// TIA Portal V17 export
// export: Created 2023-08-28T22:41:32.6164324Z, ExportSetting WithDefaults, DisplayName Totally Integrated Automation Portal, DisplayVersion V17 Update 5, DisplayName TIA Portal Openness, DisplayVersion V17 Update 5, DisplayName TIA Portal Teamcenter Gateway, DisplayVersion V17 Update 5, DisplayName TIA Portal Version Control Interface, DisplayVersion V17, DisplayName Simotion SCOUT TIA, DisplayVersion 5.4.3.0, DisplayName TIA Portal Test Suite Advanced, DisplayVersion V17 Update 1, DisplayName SIMOCODE ES, DisplayVersion V17 Update 5, DisplayName SINAMICS Startdrive Advanced, DisplayVersion V17 SP1, DisplayName SINAMICS Startdrive G130, G150, S120, S150, SINAMICS MV, S210, DisplayVersion V17 SP1, DisplayName SINAMICS Startdrive G110M, G120, G120C, G120D, G120P, G115D, DisplayVersion V17 SP1, DisplayName SIRIUS Safety ES, DisplayVersion V17 Update 5, DisplayName STEP 7 Professional, DisplayVersion V17 Update 5, DisplayName STEP 7 CFC, DisplayVersion V17 Update 1, DisplayName STEP 7 Safety, DisplayVersion V17, DisplayName WinCC Advanced, DisplayVersion V17 Update 5, DisplayName SIMATIC Visualization Architect, DisplayVersion V17 Update 5
DATA_BLOCK "FDBK_Error_n0015-uc16-el001-k30001_SN50_1"   // DB2000, F_DB
// stored: AutoNumber true, DBAccessibleFromOPCUA true, DBAccessibleFromWebserver true, InstanceOfName 03_FDBACK error, InstanceOfType FB
"03_FDBACK error "
BEGIN
END_DATA_BLOCK

DATA_BLOCK "FDBK_Error_n0015-uc16-el001-k30001_SN50_2"   // DB2001, F_DB
// stored: AutoNumber true, DBAccessibleFromOPCUA true, DBAccessibleFromWebserver true, InstanceOfName 03_FDBACK error, InstanceOfType FB
"03_FDBACK error "
BEGIN
END_DATA_BLOCK

DATA_BLOCK "FDBK_Error_n0015-uc16-el001-k30001_SN50_3"   // DB2002, F_DB
// stored: AutoNumber true, DBAccessibleFromOPCUA true, DBAccessibleFromWebserver true, InstanceOfName 03_FDBACK error, InstanceOfType FB
"03_FDBACK error "
BEGIN
END_DATA_BLOCK

DATA_BLOCK "FDBK_Error_n0017-lv004-el001-k30001_SN50_1"   // DB2003, F_DB
// stored: AutoNumber true, DBAccessibleFromOPCUA true, DBAccessibleFromWebserver true, InstanceOfName 03_FDBACK error, InstanceOfType FB
"03_FDBACK error "
BEGIN
END_DATA_BLOCK

DATA_BLOCK "FDBK_Error_n0018-lv004-el001-k30001_SN50_1"   // DB2004, F_DB
// stored: AutoNumber true, DBAccessibleFromOPCUA true, DBAccessibleFromWebserver true, InstanceOfName 03_FDBACK error, InstanceOfType FB
"03_FDBACK error "
BEGIN
END_DATA_BLOCK

DATA_BLOCK "FDBK_Error_n0020-uc15-el001-k30001_SN50_1"   // DB2005, F_DB
// stored: AutoNumber true, DBAccessibleFromOPCUA true, DBAccessibleFromWebserver true, InstanceOfName 03_FDBACK error, InstanceOfType FB
"03_FDBACK error "
BEGIN
END_DATA_BLOCK

DATA_BLOCK "FDBK_Error_n0020-uc15-el001-k30001_SN50_2"   // DB2006, F_DB
// stored: AutoNumber true, DBAccessibleFromOPCUA true, DBAccessibleFromWebserver true, InstanceOfName 03_FDBACK error, InstanceOfType FB
"03_FDBACK error "
BEGIN
END_DATA_BLOCK

DATA_BLOCK "FDBK_Error_n0020-uc15-el001-k30001_SN50_3"   // DB2007, F_DB
// stored: AutoNumber true, DBAccessibleFromOPCUA true, DBAccessibleFromWebserver true, InstanceOfName 03_FDBACK error, InstanceOfType FB
"03_FDBACK error "
BEGIN
END_DATA_BLOCK

DATA_BLOCK "FDBK_Error_n0021-icg11-el001-k30001_SN50_1"   // DB2008, F_DB
// stored: AutoNumber true, DBAccessibleFromOPCUA true, DBAccessibleFromWebserver true, InstanceOfName 03_FDBACK error, InstanceOfType FB
"03_FDBACK error "
BEGIN
END_DATA_BLOCK

DATA_BLOCK "FDBK_Error_n0022-icg21-el001-k30001_SN50_1"   // DB2009, F_DB
// stored: AutoNumber true, DBAccessibleFromOPCUA true, DBAccessibleFromWebserver true, InstanceOfName 03_FDBACK error, InstanceOfType FB
"03_FDBACK error "
BEGIN
END_DATA_BLOCK

DATA_BLOCK "FDBK_Error_n0025-uc14-el001-k30001_SN50_1"   // DB2010, F_DB
// stored: AutoNumber true, DBAccessibleFromOPCUA true, DBAccessibleFromWebserver true, InstanceOfName 03_FDBACK error, InstanceOfType FB
"03_FDBACK error "
BEGIN
END_DATA_BLOCK

DATA_BLOCK "FDBK_Error_n0025-uc14-el001-k30001_SN50_2"   // DB2011, F_DB
// stored: AutoNumber true, DBAccessibleFromOPCUA true, DBAccessibleFromWebserver true, InstanceOfName 03_FDBACK error, InstanceOfType FB
"03_FDBACK error "
BEGIN
END_DATA_BLOCK

DATA_BLOCK "FDBK_Error_n0025-uc14-el001-k30001_SN50_3"   // DB2012, F_DB
// stored: AutoNumber true, DBAccessibleFromOPCUA true, DBAccessibleFromWebserver true, InstanceOfName 03_FDBACK error, InstanceOfType FB
"03_FDBACK error "
BEGIN
END_DATA_BLOCK

DATA_BLOCK "FDBK_Error_n0039-lv001-el001-k30001_SN50_1"   // DB2013, F_DB
// stored: AutoNumber true, DBAccessibleFromOPCUA true, DBAccessibleFromWebserver true, InstanceOfName 03_FDBACK error, InstanceOfType FB
"03_FDBACK error "
BEGIN
END_DATA_BLOCK

DATA_BLOCK "FDBK_Error_n0040-lv001-el001-k30001_SN50_1"   // DB2014, F_DB
// stored: AutoNumber true, DBAccessibleFromOPCUA true, DBAccessibleFromWebserver true, InstanceOfName 03_FDBACK error, InstanceOfType FB
"03_FDBACK error "
BEGIN
END_DATA_BLOCK

DATA_BLOCK "FDBK_Error_n0041-uf31-el002-k30001_SN50_1"   // DB2015, F_DB
// stored: AutoNumber true, DBAccessibleFromOPCUA true, DBAccessibleFromWebserver true, InstanceOfName 03_FDBACK error, InstanceOfType FB
"03_FDBACK error "
BEGIN
END_DATA_BLOCK

DATA_BLOCK "FDBK_Error_n0042-uf41-el002-k30001_SN50_1"   // DB2016, F_DB
// stored: AutoNumber true, DBAccessibleFromOPCUA true, DBAccessibleFromWebserver true, InstanceOfName 03_FDBACK error, InstanceOfType FB
"03_FDBACK error "
BEGIN
END_DATA_BLOCK

DATA_BLOCK "FDBK_Error_n0044-ct1-el001-k30001_SN50_1"   // DB2017, F_DB
// stored: AutoNumber true, DBAccessibleFromOPCUA true, DBAccessibleFromWebserver true, InstanceOfName 03_FDBACK error, InstanceOfType FB
"03_FDBACK error "
BEGIN
END_DATA_BLOCK

DATA_BLOCK "FDBK_Error_n0045-ct1-el002-k30001_SN50_1"   // DB2018, F_DB
// stored: AutoNumber true, DBAccessibleFromOPCUA true, DBAccessibleFromWebserver true, InstanceOfName 03_FDBACK error, InstanceOfType FB
"03_FDBACK error "
BEGIN
END_DATA_BLOCK

DATA_BLOCK "FDBK_Error_n0046-ct1-el003-k30001_SN50_1"   // DB2019, F_DB
// stored: AutoNumber true, DBAccessibleFromOPCUA true, DBAccessibleFromWebserver true, InstanceOfName 03_FDBACK error, InstanceOfType FB
"03_FDBACK error "
BEGIN
END_DATA_BLOCK

DATA_BLOCK "FDBK_Error_n0047-lv002-el001-k30001_SN50_1"   // DB2020, F_DB
// stored: AutoNumber true, DBAccessibleFromOPCUA true, DBAccessibleFromWebserver true, InstanceOfName 03_FDBACK error, InstanceOfType FB
"03_FDBACK error "
BEGIN
END_DATA_BLOCK

DATA_BLOCK "FDBK_Error_n0048-lv002-el001-k30001_SN50_1"   // DB2021, F_DB
// stored: AutoNumber true, DBAccessibleFromOPCUA true, DBAccessibleFromWebserver true, InstanceOfName 03_FDBACK error, InstanceOfType FB
"03_FDBACK error "
BEGIN
END_DATA_BLOCK

DATA_BLOCK "FDBK_Error_n0050-uc13-el001-k30001_SN50_1"   // DB2022, F_DB
// stored: AutoNumber true, DBAccessibleFromOPCUA true, DBAccessibleFromWebserver true, InstanceOfName 03_FDBACK error, InstanceOfType FB
"03_FDBACK error "
BEGIN
END_DATA_BLOCK

DATA_BLOCK "FDBK_Error_n0050-uc13-el001-k30001_SN50_2"   // DB2023, F_DB
// stored: AutoNumber true, DBAccessibleFromOPCUA true, DBAccessibleFromWebserver true, InstanceOfName 03_FDBACK error, InstanceOfType FB
"03_FDBACK error "
BEGIN
END_DATA_BLOCK

DATA_BLOCK "FDBK_Error_n0050-uc13-el001-k30001_SN50_3"   // DB2024, F_DB
// stored: AutoNumber true, DBAccessibleFromOPCUA true, DBAccessibleFromWebserver true, InstanceOfName 03_FDBACK error, InstanceOfType FB
"03_FDBACK error "
BEGIN
END_DATA_BLOCK

DATA_BLOCK "FDBK_Error_n0053-uc12-el001-k30001_SN50_1"   // DB2025, F_DB
// stored: AutoNumber true, DBAccessibleFromOPCUA true, DBAccessibleFromWebserver true, InstanceOfName 03_FDBACK error, InstanceOfType FB
"03_FDBACK error "
BEGIN
END_DATA_BLOCK

DATA_BLOCK "FDBK_Error_n0053-uc12-el001-k30001_SN50_2"   // DB2026, F_DB
// stored: AutoNumber true, DBAccessibleFromOPCUA true, DBAccessibleFromWebserver true, InstanceOfName 03_FDBACK error, InstanceOfType FB
"03_FDBACK error "
BEGIN
END_DATA_BLOCK

DATA_BLOCK "FDBK_Error_n0053-uc12-el001-k30001_SN50_3"   // DB2027, F_DB
// stored: AutoNumber true, DBAccessibleFromOPCUA true, DBAccessibleFromWebserver true, InstanceOfName 03_FDBACK error, InstanceOfType FB
"03_FDBACK error "
BEGIN
END_DATA_BLOCK

DATA_BLOCK "FDBK_Error_n0054-uf31-el003-k30001_SN50_1"   // DB2028, F_DB
// stored: AutoNumber true, DBAccessibleFromOPCUA true, DBAccessibleFromWebserver true, InstanceOfName 03_FDBACK error, InstanceOfType FB
"03_FDBACK error "
BEGIN
END_DATA_BLOCK

DATA_BLOCK "FDBK_Error_n0057-uc11-el001-k30001_SN50_1"   // DB2029, F_DB
// stored: AutoNumber true, DBAccessibleFromOPCUA true, DBAccessibleFromWebserver true, InstanceOfName 03_FDBACK error, InstanceOfType FB
"03_FDBACK error "
BEGIN
END_DATA_BLOCK

DATA_BLOCK "FDBK_Error_n0057-uc11-el001-k30001_SN50_2"   // DB2030, F_DB
// stored: AutoNumber true, DBAccessibleFromOPCUA true, DBAccessibleFromWebserver true, InstanceOfName 03_FDBACK error, InstanceOfType FB
"03_FDBACK error "
BEGIN
END_DATA_BLOCK

DATA_BLOCK "FDBK_Error_n0057-uc11-el001-k30001_SN50_3"   // DB2031, F_DB
// stored: AutoNumber true, DBAccessibleFromOPCUA true, DBAccessibleFromWebserver true, InstanceOfName 03_FDBACK error, InstanceOfType FB
"03_FDBACK error "
BEGIN
END_DATA_BLOCK

DATA_BLOCK "FDBK_Error_n0058-lv003-el001-k30001_SN50_1"   // DB2032, F_DB
// stored: AutoNumber true, DBAccessibleFromOPCUA true, DBAccessibleFromWebserver true, InstanceOfName 03_FDBACK error, InstanceOfType FB
"03_FDBACK error "
BEGIN
END_DATA_BLOCK

DATA_BLOCK "FDBK_Error_n0059-lv003-el001-k30001_SN50_1"   // DB2033, F_DB
// stored: AutoNumber true, DBAccessibleFromOPCUA true, DBAccessibleFromWebserver true, InstanceOfName 03_FDBACK error, InstanceOfType FB
"03_FDBACK error "
BEGIN
END_DATA_BLOCK

DATA_BLOCK "FDBK_Error_n0028-uc17-el001-k30001_SN50_1"   // DB2034, F_DB
// stored: AutoNumber true, DBAccessibleFromOPCUA true, DBAccessibleFromWebserver true, InstanceOfName 03_FDBACK error, InstanceOfType FB
"03_FDBACK error "
BEGIN
END_DATA_BLOCK

DATA_BLOCK "FDBK_Error_n0028-uc17-el001-k30001_SN50_2"   // DB2035, F_DB
// stored: AutoNumber true, DBAccessibleFromOPCUA true, DBAccessibleFromWebserver true, InstanceOfName 03_FDBACK error, InstanceOfType FB
"03_FDBACK error "
BEGIN
END_DATA_BLOCK

DATA_BLOCK "FDBK_Error_n0033-zp001-el001-k40001_SN50_1"   // DB2036, F_DB
// stored: AutoNumber true, DBAccessibleFromOPCUA true, DBAccessibleFromWebserver true, InstanceOfName 03_FDBACK error, InstanceOfType FB
"03_FDBACK error "
BEGIN
END_DATA_BLOCK

DATA_BLOCK "FDBK_Error_n0033-zp001-el001-k40001_SN50_2"   // DB2037, F_DB
// stored: AutoNumber true, DBAccessibleFromOPCUA true, DBAccessibleFromWebserver true, InstanceOfName 03_FDBACK error, InstanceOfType FB
"03_FDBACK error "
BEGIN
END_DATA_BLOCK

DATA_BLOCK "FDBK_Error_n0034-ug6-el001-k30001_SN50_1"   // DB2038, F_DB
// stored: AutoNumber true, DBAccessibleFromOPCUA true, DBAccessibleFromWebserver true, InstanceOfName 03_FDBACK error, InstanceOfType FB
"03_FDBACK error "
BEGIN
END_DATA_BLOCK

DATA_BLOCK "FDBK_Error_n0034-ug6-el001-k30001_SN50_2"   // DB2039, F_DB
// stored: AutoNumber true, DBAccessibleFromOPCUA true, DBAccessibleFromWebserver true, InstanceOfName 03_FDBACK error, InstanceOfType FB
"03_FDBACK error "
BEGIN
END_DATA_BLOCK

DATA_BLOCK "FDBK_Error_n0034-ug6-el001-k30001_SN50_3"   // DB2040, F_DB
// stored: AutoNumber true, DBAccessibleFromOPCUA true, DBAccessibleFromWebserver true, InstanceOfName 03_FDBACK error, InstanceOfType FB
"03_FDBACK error "
BEGIN
END_DATA_BLOCK

DATA_BLOCK "FDBK_Error_n0043-db93-el001-k30001_SN50_1"   // DB2041, F_DB
// stored: AutoNumber true, DBAccessibleFromOPCUA true, DBAccessibleFromWebserver true, InstanceOfName 03_FDBACK error, InstanceOfType FB
"03_FDBACK error "
BEGIN
END_DATA_BLOCK

DATA_BLOCK "FDBK_Error_n0005-lv008-el001-k30001_SN51_1"   // DB2042, F_DB
// stored: AutoNumber true, DBAccessibleFromOPCUA true, DBAccessibleFromWebserver true, InstanceOfName 03_FDBACK error, InstanceOfType FB
"03_FDBACK error "
BEGIN
END_DATA_BLOCK

DATA_BLOCK "FDBK_Error_n0006-lv008-el001-k30001_SN51_1"   // DB2043, F_DB
// stored: AutoNumber true, DBAccessibleFromOPCUA true, DBAccessibleFromWebserver true, InstanceOfName 03_FDBACK error, InstanceOfType FB
"03_FDBACK error "
BEGIN
END_DATA_BLOCK

DATA_BLOCK "FDBK_Error_n0007-icg22-el001-k30001_SN51_1"   // DB2044, F_DB
// stored: AutoNumber true, DBAccessibleFromOPCUA true, DBAccessibleFromWebserver true, InstanceOfName 03_FDBACK error, InstanceOfType FB
"03_FDBACK error "
BEGIN
END_DATA_BLOCK

DATA_BLOCK "FDBK_Error_n0008-icg12-el001-k30001_SN51_1"   // DB2045, F_DB
// stored: AutoNumber true, DBAccessibleFromOPCUA true, DBAccessibleFromWebserver true, InstanceOfName 03_FDBACK error, InstanceOfType FB
"03_FDBACK error "
BEGIN
END_DATA_BLOCK

DATA_BLOCK "FDBK_Error_n0009-uf42-el002-k30001_SN51_1"   // DB2046, F_DB
// stored: AutoNumber true, DBAccessibleFromOPCUA true, DBAccessibleFromWebserver true, InstanceOfName 03_FDBACK error, InstanceOfType FB
"03_FDBACK error "
BEGIN
END_DATA_BLOCK

DATA_BLOCK "FDBK_Error_n0010-lv007-el001-k30001_SN51_1"   // DB2047, F_DB
// stored: AutoNumber true, DBAccessibleFromOPCUA true, DBAccessibleFromWebserver true, InstanceOfName 03_FDBACK error, InstanceOfType FB
"03_FDBACK error "
BEGIN
END_DATA_BLOCK

DATA_BLOCK "FDBK_Error_n0011-lv007-el001-k30001_SN51_1"   // DB2048, F_DB
// stored: AutoNumber true, DBAccessibleFromOPCUA true, DBAccessibleFromWebserver true, InstanceOfName 03_FDBACK error, InstanceOfType FB
"03_FDBACK error "
BEGIN
END_DATA_BLOCK

DATA_BLOCK "FDBK_Error_n0025-dc91-el001-k30001_SN51_1"   // DB2049, F_DB
// stored: AutoNumber true, DBAccessibleFromOPCUA true, DBAccessibleFromWebserver true, InstanceOfName 03_FDBACK error, InstanceOfType FB
"03_FDBACK error "
BEGIN
END_DATA_BLOCK

DATA_BLOCK "FDBK_Error_n0028-lv005-el001-k30001_SN51_1"   // DB2050, F_DB
// stored: AutoNumber true, DBAccessibleFromOPCUA true, DBAccessibleFromWebserver true, InstanceOfName 03_FDBACK error, InstanceOfType FB
"03_FDBACK error "
BEGIN
END_DATA_BLOCK

DATA_BLOCK "FDBK_Error_n0029-ct2-el001-k30001_SN51_1"   // DB2051, F_DB
// stored: AutoNumber true, DBAccessibleFromOPCUA true, DBAccessibleFromWebserver true, InstanceOfName 03_FDBACK error, InstanceOfType FB
"03_FDBACK error "
BEGIN
END_DATA_BLOCK

DATA_BLOCK "FDBK_Error_n0033-uc26-el001-k30001_SN51_1"   // DB2052, F_DB
// stored: AutoNumber true, DBAccessibleFromOPCUA true, DBAccessibleFromWebserver true, InstanceOfName 03_FDBACK error, InstanceOfType FB
"03_FDBACK error "
BEGIN
END_DATA_BLOCK

DATA_BLOCK "FDBK_Error_n0033-uc26-el001-k30001_SN51_2"   // DB2053, F_DB
// stored: AutoNumber true, DBAccessibleFromOPCUA true, DBAccessibleFromWebserver true, InstanceOfName 03_FDBACK error, InstanceOfType FB
"03_FDBACK error "
BEGIN
END_DATA_BLOCK

DATA_BLOCK "FDBK_Error_n0033-uc26-el001-k30001_SN51_3"   // DB2054, F_DB
// stored: AutoNumber true, DBAccessibleFromOPCUA true, DBAccessibleFromWebserver true, InstanceOfName 03_FDBACK error, InstanceOfType FB
"03_FDBACK error "
BEGIN
END_DATA_BLOCK

DATA_BLOCK "FDBK_Error_n0035-ct2-el002-k30001_SN51_1"   // DB2055, F_DB
// stored: AutoNumber true, DBAccessibleFromOPCUA true, DBAccessibleFromWebserver true, InstanceOfName 03_FDBACK error, InstanceOfType FB
"03_FDBACK error "
BEGIN
END_DATA_BLOCK

DATA_BLOCK "FDBK_Error_n0036-lv005-el001-k30001_SN51_1"   // DB2056, F_DB
// stored: AutoNumber true, DBAccessibleFromOPCUA true, DBAccessibleFromWebserver true, InstanceOfName 03_FDBACK error, InstanceOfType FB
"03_FDBACK error "
BEGIN
END_DATA_BLOCK

DATA_BLOCK "FDBK_Error_n0041-uc27-el001-k30001_SN51_1"   // DB2057, F_DB
// stored: AutoNumber true, DBAccessibleFromOPCUA true, DBAccessibleFromWebserver true, InstanceOfName 03_FDBACK error, InstanceOfType FB
"03_FDBACK error "
BEGIN
END_DATA_BLOCK

DATA_BLOCK "FDBK_Error_n0041-uc27-el001-k30001_SN51_2"   // DB2058, F_DB
// stored: AutoNumber true, DBAccessibleFromOPCUA true, DBAccessibleFromWebserver true, InstanceOfName 03_FDBACK error, InstanceOfType FB
"03_FDBACK error "
BEGIN
END_DATA_BLOCK

DATA_BLOCK "FDBK_Error_n0046-uc25-el001-k30001_SN51_1"   // DB2059, F_DB
// stored: AutoNumber true, DBAccessibleFromOPCUA true, DBAccessibleFromWebserver true, InstanceOfName 03_FDBACK error, InstanceOfType FB
"03_FDBACK error "
BEGIN
END_DATA_BLOCK

DATA_BLOCK "FDBK_Error_n0046-uc25-el001-k30001_SN51_2"   // DB2060, F_DB
// stored: AutoNumber true, DBAccessibleFromOPCUA true, DBAccessibleFromWebserver true, InstanceOfName 03_FDBACK error, InstanceOfType FB
"03_FDBACK error "
BEGIN
END_DATA_BLOCK

DATA_BLOCK "FDBK_Error_n0046-uc25-el001-k30001_SN51_3"   // DB2061, F_DB
// stored: AutoNumber true, DBAccessibleFromOPCUA true, DBAccessibleFromWebserver true, InstanceOfName 03_FDBACK error, InstanceOfType FB
"03_FDBACK error "
BEGIN
END_DATA_BLOCK

DATA_BLOCK "FDBK_Error_n0048-lv006-el001-k30001_SN51_1"   // DB2062, F_DB
// stored: AutoNumber true, DBAccessibleFromOPCUA true, DBAccessibleFromWebserver true, InstanceOfName 03_FDBACK error, InstanceOfType FB
"03_FDBACK error "
BEGIN
END_DATA_BLOCK

DATA_BLOCK "FDBK_Error_n0051-uc24-el001-k30001_SN51_1"   // DB2063, F_DB
// stored: AutoNumber true, DBAccessibleFromOPCUA true, DBAccessibleFromWebserver true, InstanceOfName 03_FDBACK error, InstanceOfType FB
"03_FDBACK error "
BEGIN
END_DATA_BLOCK

DATA_BLOCK "FDBK_Error_n0051-uc24-el001-k30001_SN51_2"   // DB2064, F_DB
// stored: AutoNumber true, DBAccessibleFromOPCUA true, DBAccessibleFromWebserver true, InstanceOfName 03_FDBACK error, InstanceOfType FB
"03_FDBACK error "
BEGIN
END_DATA_BLOCK

DATA_BLOCK "FDBK_Error_n0051-uc24-el001-k30001_SN51_3"   // DB2065, F_DB
// stored: AutoNumber true, DBAccessibleFromOPCUA true, DBAccessibleFromWebserver true, InstanceOfName 03_FDBACK error, InstanceOfType FB
"03_FDBACK error "
BEGIN
END_DATA_BLOCK

DATA_BLOCK "FDBK_Error_n0056-uc23-el001-k30001_SN51_1"   // DB2066, F_DB
// stored: AutoNumber true, DBAccessibleFromOPCUA true, DBAccessibleFromWebserver true, InstanceOfName 03_FDBACK error, InstanceOfType FB
"03_FDBACK error "
BEGIN
END_DATA_BLOCK

DATA_BLOCK "FDBK_Error_n0056-uc23-el001-k30001_SN51_2"   // DB2067, F_DB
// stored: AutoNumber true, DBAccessibleFromOPCUA true, DBAccessibleFromWebserver true, InstanceOfName 03_FDBACK error, InstanceOfType FB
"03_FDBACK error "
BEGIN
END_DATA_BLOCK

DATA_BLOCK "FDBK_Error_n0056-uc23-el001-k30001_SN51_3"   // DB2068, F_DB
// stored: AutoNumber true, DBAccessibleFromOPCUA true, DBAccessibleFromWebserver true, InstanceOfName 03_FDBACK error, InstanceOfType FB
"03_FDBACK error "
BEGIN
END_DATA_BLOCK

DATA_BLOCK "FDBK_Error_n0058-ct2-el003-k30001_SN51_1"   // DB2069, F_DB
// stored: AutoNumber true, DBAccessibleFromOPCUA true, DBAccessibleFromWebserver true, InstanceOfName 03_FDBACK error, InstanceOfType FB
"03_FDBACK error "
BEGIN
END_DATA_BLOCK

DATA_BLOCK "FDBK_Error_n0061-uc22-el001-k30001_SN51_1"   // DB2070, F_DB
// stored: AutoNumber true, DBAccessibleFromOPCUA true, DBAccessibleFromWebserver true, InstanceOfName 03_FDBACK error, InstanceOfType FB
"03_FDBACK error "
BEGIN
END_DATA_BLOCK

DATA_BLOCK "FDBK_Error_n0061-uc22-el001-k30001_SN51_2"   // DB2071, F_DB
// stored: AutoNumber true, DBAccessibleFromOPCUA true, DBAccessibleFromWebserver true, InstanceOfName 03_FDBACK error, InstanceOfType FB
"03_FDBACK error "
BEGIN
END_DATA_BLOCK

DATA_BLOCK "FDBK_Error_n0061-uc22-el001-k30001_SN51_3"   // DB2072, F_DB
// stored: AutoNumber true, DBAccessibleFromOPCUA true, DBAccessibleFromWebserver true, InstanceOfName 03_FDBACK error, InstanceOfType FB
"03_FDBACK error "
BEGIN
END_DATA_BLOCK

DATA_BLOCK "FDBK_Error_n0063-lv006-el001-k30001_SN51_1"   // DB2073, F_DB
// stored: AutoNumber true, DBAccessibleFromOPCUA true, DBAccessibleFromWebserver true, InstanceOfName 03_FDBACK error, InstanceOfType FB
"03_FDBACK error "
BEGIN
END_DATA_BLOCK

DATA_BLOCK "FDBK_Error_n0066-uc21-el001-k30001_SN51_1"   // DB2074, F_DB
// stored: AutoNumber true, DBAccessibleFromOPCUA true, DBAccessibleFromWebserver true, InstanceOfName 03_FDBACK error, InstanceOfType FB
"03_FDBACK error "
BEGIN
END_DATA_BLOCK

DATA_BLOCK "FDBK_Error_n0066-uc21-el001-k30001_SN51_2"   // DB2075, F_DB
// stored: AutoNumber true, DBAccessibleFromOPCUA true, DBAccessibleFromWebserver true, InstanceOfName 03_FDBACK error, InstanceOfType FB
"03_FDBACK error "
BEGIN
END_DATA_BLOCK

DATA_BLOCK "FDBK_Error_n0066-uc21-el001-k30001_SN51_3"   // DB2076, F_DB
// stored: AutoNumber true, DBAccessibleFromOPCUA true, DBAccessibleFromWebserver true, InstanceOfName 03_FDBACK error, InstanceOfType FB
"03_FDBACK error "
BEGIN
END_DATA_BLOCK

DATA_BLOCK "FDBK_Error_n0070-uf31-el001-k30001_SN51_1"   // DB2077, F_DB
// stored: AutoNumber true, DBAccessibleFromOPCUA true, DBAccessibleFromWebserver true, InstanceOfName 03_FDBACK error, InstanceOfType FB
"03_FDBACK error "
BEGIN
END_DATA_BLOCK

DATA_BLOCK "FDBK_Error_n0071-uf41-el001-k30001_SN51_1"   // DB2078, F_DB
// stored: AutoNumber true, DBAccessibleFromOPCUA true, DBAccessibleFromWebserver true, InstanceOfName 03_FDBACK error, InstanceOfType FB
"03_FDBACK error "
BEGIN
END_DATA_BLOCK

DATA_BLOCK "FDBK_Error_n0072-uf51-el001-k30001_SN51_1"   // DB2079, F_DB
// stored: AutoNumber true, DBAccessibleFromOPCUA true, DBAccessibleFromWebserver true, InstanceOfName 03_FDBACK error, InstanceOfType FB
"03_FDBACK error "
BEGIN
END_DATA_BLOCK

DATA_BLOCK "FDBK_Error_n0073-ifg31-el001-k30001_SN51_1"   // DB2080, F_DB
// stored: AutoNumber true, DBAccessibleFromOPCUA true, DBAccessibleFromWebserver true, InstanceOfName 03_FDBACK error, InstanceOfType FB
"03_FDBACK error "
BEGIN
END_DATA_BLOCK

DATA_BLOCK "FDBK_Error_n0074-ifg41-el001-k30001_SN51_1"   // DB2081, F_DB
// stored: AutoNumber true, DBAccessibleFromOPCUA true, DBAccessibleFromWebserver true, InstanceOfName 03_FDBACK error, InstanceOfType FB
"03_FDBACK error "
BEGIN
END_DATA_BLOCK

DATA_BLOCK "FDBK_Error_n0075-uf32-el001-k30001_SN51_1"   // DB2082, F_DB
// stored: AutoNumber true, DBAccessibleFromOPCUA true, DBAccessibleFromWebserver true, InstanceOfName 03_FDBACK error, InstanceOfType FB
"03_FDBACK error "
BEGIN
END_DATA_BLOCK

DATA_BLOCK "FDBK_Error_n0076-uf42-el001-k30001_SN51_1"   // DB2083, F_DB
// stored: AutoNumber true, DBAccessibleFromOPCUA true, DBAccessibleFromWebserver true, InstanceOfName 03_FDBACK error, InstanceOfType FB
"03_FDBACK error "
BEGIN
END_DATA_BLOCK

DATA_BLOCK "FDBK_Error_n0082-zp002-el001-k30001_SN51_1"   // DB2084, F_DB
// stored: AutoNumber true, DBAccessibleFromOPCUA true, DBAccessibleFromWebserver true, InstanceOfName 03_FDBACK error, InstanceOfType FB
"03_FDBACK error "
BEGIN
END_DATA_BLOCK

DATA_BLOCK "FDBK_Error_n0083-lv001-el001-k30001_SN51_1"   // DB2085, F_DB
// stored: AutoNumber true, DBAccessibleFromOPCUA true, DBAccessibleFromWebserver true, InstanceOfName 03_FDBACK error, InstanceOfType FB
"03_FDBACK error "
BEGIN
END_DATA_BLOCK

DATA_BLOCK "FDBK_Error_n0084-lv001-el001-k30001_SN51_1"   // DB2086, F_DB
// stored: AutoNumber true, DBAccessibleFromOPCUA true, DBAccessibleFromWebserver true, InstanceOfName 03_FDBACK error, InstanceOfType FB
"03_FDBACK error "
BEGIN
END_DATA_BLOCK

DATA_BLOCK "FDBK_Error_n0085-uc29-el001-k30001_SN51_1"   // DB2087, F_DB
// stored: AutoNumber true, DBAccessibleFromOPCUA true, DBAccessibleFromWebserver true, InstanceOfName 03_FDBACK error, InstanceOfType FB
"03_FDBACK error "
BEGIN
END_DATA_BLOCK

DATA_BLOCK "FDBK_Error_n0091-zp001-el001-k30001_SN51_1"   // DB2088, F_DB
// stored: AutoNumber true, DBAccessibleFromOPCUA true, DBAccessibleFromWebserver true, InstanceOfName 03_FDBACK error, InstanceOfType FB
"03_FDBACK error "
BEGIN
END_DATA_BLOCK

DATA_BLOCK "FDBK_Error_n0091-zp001-el001-k30001_SN51_2"   // DB2089, F_DB
// stored: AutoNumber true, DBAccessibleFromOPCUA true, DBAccessibleFromWebserver true, InstanceOfName 03_FDBACK error, InstanceOfType FB
"03_FDBACK error "
BEGIN
END_DATA_BLOCK

DATA_BLOCK "FDBK_Error_n0093-ug7-el001-k30001_SN51_1"   // DB2090, F_DB
// stored: AutoNumber true, DBAccessibleFromOPCUA true, DBAccessibleFromWebserver true, InstanceOfName 03_FDBACK error, InstanceOfType FB
"03_FDBACK error "
BEGIN
END_DATA_BLOCK

DATA_BLOCK "FDBK_Error_n0093-ug7-el001-k30001_SN51_2"   // DB2091, F_DB
// stored: AutoNumber true, DBAccessibleFromOPCUA true, DBAccessibleFromWebserver true, InstanceOfName 03_FDBACK error, InstanceOfType FB
"03_FDBACK error "
BEGIN
END_DATA_BLOCK

DATA_BLOCK "FDBK_Error_n0093-ug7-el001-k30001_SN51_3"   // DB2092, F_DB
// stored: AutoNumber true, DBAccessibleFromOPCUA true, DBAccessibleFromWebserver true, InstanceOfName 03_FDBACK error, InstanceOfType FB
"03_FDBACK error "
BEGIN
END_DATA_BLOCK
